// SIMATIC S7-200 project (STEP 7-Micro/WIN), CPU 222 REL 02.01

SYMBOL_TABLE USER1
P_SALITA         I0.0     // PULSANTE SALITA
P_DISCESA        I0.1     // PULSANTE DISCESA
P_STOP           I0.2     // PULSANTE DI ARRESTO
FC_SUP           I0.3     // FINECORSA SUPERIORE
FC_INF           I0.4     // FINECORSA INFERIORE
SALITA           Q0.0     // COMANDO DI SALITA
DISCESA          Q0.1     // COMANDO DISCESA
END_SYMBOL_TABLE

ORGANIZATION_BLOCK MAIN:OB1
TITLE=DPS 203 MONTACARICHI
BEGIN
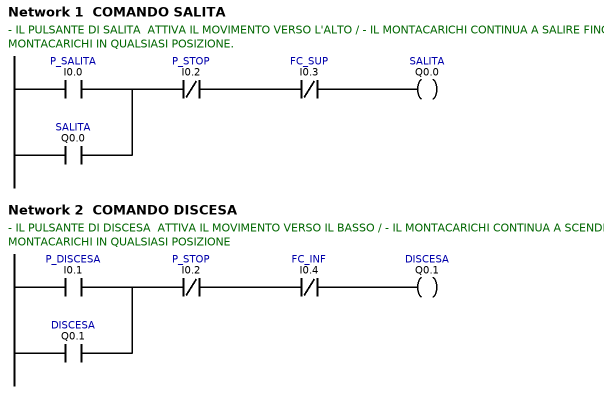
Network 1 // COMANDO SALITA 
// - IL PULSANTE DI SALITA  ATTIVA IL MOVIMENTO VERSO L'ALTO
// - IL MONTACARICHI CONTINUA A SALIRE FINO AL' INTERVENTO DEL FC_SUP
// - IL PULSANTE DI STOP ARRESTA LA SALITA DEL  MONTACARICHI IN QUALSIASI POSIZIONE.
LD     P_SALITA:I0.0
O      SALITA:Q0.0
AN     P_STOP:I0.2
AN     FC_SUP:I0.3
=      SALITA:Q0.0
Network 2 // COMANDO DISCESA
// - IL PULSANTE DI DISCESA  ATTIVA IL MOVIMENTO VERSO IL BASSO
// - IL MONTACARICHI CONTINUA A SCENDERE FINO AL' INTERVENTO DEL FC_INF
// - IL PULSANTE DI STOP ARRESTA LA DISCESA  DEL  MONTACARICHI IN QUALSIASI POSIZIONE
LD     P_DISCESA:I0.1
O      DISCESA:Q0.1
AN     P_STOP:I0.2
AN     FC_INF:I0.4
=      DISCESA:Q0.1
END_ORGANIZATION_BLOCK
